PROGRAM MAIN
VAR
	axis: AXIS_REF;
	iTermBits: INT;
	rV : Real;
	i_iDistance_R AT %I* :INT;
	rVref : Real;
	i_irefV_R AT %I* :INT;
	power: MC_POWER;
	retracted AT %I* : BOOL;
	extended At %I* :BOOL;
END_VAR

//axis.ReadStatus();
iTermBits := 32767;
rV := 10*INT_TO_REAL(i_iDistance_R)/iTermBits;
rVref := 10*INT_TO_REAL(i_irefV_R)/iTermBits;
//retracted limit switch is the one close to the motork drive, both limit switches are NO
// Retract is the postive direction, extend is negative  
power(Axis:=axis, Enable_Positive := NOT retracted, Enable_Negative:= NOT extended);

END_PROGRAM

(* stored: Version 1.1.0.1, ProductVersion 3.1.4022.18
   POU MAIN: Id {19271f00-77b4-42b9-839b-a8810c343e66}, SpecialFunc None *)
